(* IEC 61131-3 sources: controlforge-structured-text/manual-tests/code-actions, 5 files *)

(* ---- missing-end-blocks.st ---- *)
(* Test: Missing END_* blocks - should show code actions to insert missing closing keywords *)

PROGRAM Main
VAR
    x : INT;
END_VAR
    IF x > 0 THEN
        x := 10;
(* Missing END_IF - should offer quick fix to insert it *)

FUNCTION Add : INT
VAR_INPUT
    a : INT;
    b : INT;
END_VAR
    Add := a + b;
(* Missing END_FUNCTION - should offer quick fix *)

FUNCTION_BLOCK FB_Motor
VAR_INPUT
    start : BOOL;
END_VAR
VAR_OUTPUT
    running : BOOL;
(* Missing END_VAR - should offer quick fix *)
(* Missing END_FUNCTION_BLOCK - should offer quick fix *)

(* ---- missing-declaration.st ---- *)
// Manual test: Missing Variable Declaration Detection & Auto-Fix
//
// How to test:
//  1. Open this file in VS Code with ControlForge ST extension active.
//  2. The undefined variables below will show yellow squiggles.
//  3. Hover over each squiggle or click the light bulb (Ctrl+.) to see quick fixes.
//
// Expected quick-fix actions per variable:
//  - undeclaredBool  → "Declare 'undeclaredBool' as BOOL"
//  - undeclaredInt   → "Declare 'undeclaredInt' as INT"
//  - undeclaredReal  → "Declare 'undeclaredReal' as REAL"
//  - undeclaredTime  → "Declare 'undeclaredTime' as TIME"
//  - undeclaredStr   → "Declare 'undeclaredStr' as STRING"
//  - myTimer         → "Declare 'myTimer' as TON"
//  - myCounter       → "Declare 'myCounter' as CTU"
//
// When there are multiple undefined vars, an additional batch action appears:
//  - "Declare all N undefined variables"
//
// After applying a fix, the new declaration should appear inside the VAR block
// and the squiggle should disappear.

PROGRAM MissingDeclarationTest
VAR
    existingVar : INT := 0;
END_VAR

    // BOOL — assigned TRUE/FALSE
    undeclaredBool := TRUE;

    // INT — assigned integer literal
    undeclaredInt := 100;

    // REAL — assigned float literal
    undeclaredReal := 3.14;

    // TIME — assigned T# literal
    undeclaredTime := T#10s;

    // STRING — assigned string literal
    undeclaredStr := 'hello world';

    // TON instance — member access .Q and .ET
    myTimer(IN := existingVar > 0, PT := T#5s);
    IF myTimer.Q THEN
        existingVar := myTimer.ET;
    END_IF

    // CTU instance — member access .CV
    myCounter(CU := undeclaredBool, R := FALSE, PV := 10);
    existingVar := myCounter.CV;

END_PROGRAM

// Test: no local VAR block — fix should create one
PROGRAM NoPriorVarBlock
VAR_INPUT
    trigger : BOOL;
END_VAR

    // undeclaredLocal should get a new VAR block inserted
    undeclaredLocal := 99;

END_PROGRAM

(* ---- orphaned-ends.st ---- *)
(* Test: Orphaned END_* keywords - should show code actions to remove them *)

END_PROGRAM
(* Orphaned END_PROGRAM without opener - should offer quick fix to remove *)

PROGRAM Main
VAR
    x : INT;
END_VAR
    END_IF
(* Orphaned END_IF without matching IF - should offer quick fix to remove *)

    END_VAR
(* Orphaned END_VAR - should offer quick fix to remove *)
END_PROGRAM

(* ---- unclosed-strings.st ---- *)
(* Test: Unclosed string literals - should show code actions to close them *)

PROGRAM Main
VAR
    msg1 : STRING := 'Hello World;
(* Missing closing single quote - should offer quick fix *)

    msg2 : WSTRING := "Wide String;
(* Missing closing double quote - should offer quick fix *)

    msg3 : STRING := 'Test;
(* Should insert quote before semicolon *)
END_VAR
END_PROGRAM

(* ---- unmatched-parens.st ---- *)
(* Test: Unmatched parentheses - should show code actions to fix them *)

PROGRAM Main
VAR
    x : INT;
    y : REAL;
END_VAR
    x := (1 + 2;
(* Missing closing paren - should offer quick fix to add ) *)

    y := ((3.0 * 4.0;
(* Two missing closing parens - should offer quick fix to add )) *)

    x := 5 + 6);
(* Extra closing paren - should offer quick fix to remove *)
END_PROGRAM
